FUNCTION_BLOCK HeatPumpController2 (* Simple SG Ready heat pump controller for battery systems *)
  (* Standard: 61499-2; Description: Sets the output to NORMAL (0:0) if there are no PV surpluses. If there are surpluses, the output is set to AMPLIFIED (0:1). *)
  (* Version 1.0, 2017-07-29, Marc Jakobi, HTW Berlin *)
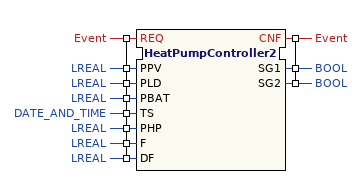
  EVENT_INPUT
    REQ WITH PLD, PPV, PBAT, PHP, F, TS, DF; (* Normal Execution Request *)
  END_EVENT
  EVENT_OUTPUT
    CNF WITH SG1, SG2; (* Execution Confirmation *)
  END_EVENT
  VAR_INPUT
    PPV : LREAL; (* PV power in W *)
    PLD : LREAL; (* Load in W *)
    PBAT : LREAL; (* Battery charging power in W *)
    TS : DATE_AND_TIME; (* Time stamp *)
    PHP : LREAL; (* Heat pump's nominal electrical power in kW *)
    F : LREAL := 1; (* On/Off threshold [0.1,..,1] *)
    DF : LREAL; (* Derating factor for the PV system [0,..,1] *)
  END_VAR
  VAR_OUTPUT
    SG1 : BOOL; (* SG Ready output 1 *)
    SG2 : BOOL; (* SG Ready output 2 *)
  END_VAR
  FBS
    FB_PVFEEDIN_CALC : FB_PVFEEDIN_CALC;
    F_LIMIT : F_LIMIT(MN := LREAL#0.1, MX := LREAL#1.5);
    HIGH_KW : F_MUL;
    MEAN_PV_W : F_N_MIN_MEAN_LREAL(N := T#1m);
    MEAN_LOAD_W : F_N_MIN_MEAN_LREAL(N := T#1m);
    MEAN_BAT_W : F_N_MIN_MEAN_LREAL(N := T#1m);
    E_MERGE : E_MERGE;
    E_MERGE_1 : E_MERGE;
    F : LREAL2LREAL;
    LOW_W : F_MUL;
    SWITCH_STATE : F_OR;
    BOOL2BOOL_1 : BOOL2BOOL;
    E_SWITCH : E_SWITCH;
    E_MERGE_2 : E_MERGE;
    E_MERGE_3 : E_MERGE;
    HIGH_W : F_MUL(IN2 := LREAL#1000);
    C_HIGH_KW : LREAL2LREAL;
    C_HIGH_W : LREAL2LREAL;
    C_LOW_W : LREAL2LREAL;
    NORMAL : F_LE;
    AMPLIFIED : F_GE;
    F_LT : F_LT(IN2 := LREAL#1);
    F_SEL : F_SEL(IN0 := BOOL#0, IN1 := BOOL#1);
  END_FBS
  EVENT_CONNECTIONS
    REQ TO MEAN_PV_W.REQ;
    MEAN_PV_W.CNF1 TO E_MERGE.EI1;
    MEAN_PV_W.CNF0 TO E_MERGE.EI2;
    E_MERGE.EO TO MEAN_LOAD_W.REQ;
    MEAN_LOAD_W.CNF1 TO E_MERGE_1.EI1;
    MEAN_LOAD_W.CNF0 TO E_MERGE_1.EI2;
    E_MERGE_1.EO TO MEAN_BAT_W.REQ;
    MEAN_BAT_W.CNF1 TO F_LIMIT.REQ;
    F_LIMIT.CNF TO F.REQ;
    F.CNF TO HIGH_KW.REQ;
    SWITCH_STATE.CNF TO E_SWITCH.EI;
    BOOL2BOOL_1.CNF TO E_MERGE_2.EI1;
    E_SWITCH.EO0 TO E_MERGE_2.EI2;
    E_MERGE_2.EO TO E_MERGE_3.EI1;
    MEAN_BAT_W.CNF0 TO E_MERGE_3.EI2;
    HIGH_KW.CNF TO C_HIGH_KW.REQ;
    C_HIGH_KW.CNF TO HIGH_W.REQ;
    HIGH_W.CNF TO C_HIGH_W.REQ;
    C_HIGH_W.CNF TO LOW_W.REQ;
    LOW_W.CNF TO C_LOW_W.REQ;
    C_LOW_W.CNF TO FB_PVFEEDIN_CALC.REQ;
    NORMAL.CNF TO SWITCH_STATE.REQ;
    FB_PVFEEDIN_CALC.CNF TO AMPLIFIED.REQ;
    AMPLIFIED.CNF TO NORMAL.REQ;
    E_SWITCH.EO1 TO F_LT.REQ;
    F_LT.CNF TO F_SEL.REQ;
    F_SEL.CNF TO BOOL2BOOL_1.REQ;
    E_MERGE_3.EO TO CNF;
  END_CONNECTIONS
  DATA_CONNECTIONS
    F TO F_LIMIT.IN;
    TS TO MEAN_PV_W.TSI;
    PPV TO MEAN_PV_W.X;
    TS TO MEAN_LOAD_W.TSI;
    PLD TO MEAN_LOAD_W.X;
    PBAT TO MEAN_BAT_W.X;
    TS TO MEAN_BAT_W.TSI;
    MEAN_PV_W.Y TO FB_PVFEEDIN_CALC.PPV;
    MEAN_LOAD_W.Y TO FB_PVFEEDIN_CALC.PLD;
    MEAN_BAT_W.Y TO FB_PVFEEDIN_CALC.PBAT;
    F_LIMIT.OUT TO F.IN;
    PHP TO HIGH_KW.IN2;
    F.OUT TO HIGH_KW.IN1;
    F.OUT TO LOW_W.IN2;
    MEAN_LOAD_W.Y TO LOW_W.IN1;
    BOOL2BOOL_1.OUT TO SG2;
    SWITCH_STATE.OUT TO E_SWITCH.G;
    HIGH_KW.OUT TO C_HIGH_KW.IN;
    C_HIGH_KW.OUT TO HIGH_W.IN1;
    HIGH_W.OUT TO C_HIGH_W.IN;
    LOW_W.OUT TO C_LOW_W.IN;
    MEAN_PV_W.Y TO NORMAL.IN1;
    C_LOW_W.OUT TO NORMAL.IN2;
    NORMAL.OUT TO SWITCH_STATE.IN2;
    FB_PVFEEDIN_CALC.PGF TO AMPLIFIED.IN1;
    C_HIGH_W.OUT TO AMPLIFIED.IN2;
    AMPLIFIED.OUT TO SWITCH_STATE.IN1;
    AMPLIFIED.OUT TO BOOL2BOOL_1.IN;
    DF TO F_LT.IN1;
    F_LT.OUT TO F_SEL.G;
    F_SEL.OUT TO SG1;
  END_CONNECTIONS
END_FUNCTION_BLOCK
